Universal Robots PolyScope program: socketbuffer.urp

Program socketbuffer (installation=botross directory=/programs/APS2OsUltimosRomanticos createdIn=3.15.3.106223 lastSavedIn=3.15.3.106223 robotSerialNumber=2017357017)
Calibrated DH parameters: a=[0.0001, -0.032836, -0.39033, 0.000086, 0.000053, 0]; d=[0.089393, 264.548863, -261.578988, -2.85966, 0.094927, 0.082356]; alpha=[1.569373, -0.001603, 0.013671, 1.570599, -1.570158, 0]; deltaTheta=[0.000031, -1.49356, 1.597104, -0.103695, -0.000023, -0.000043]
Robot Program (runOnlyOnce=false)
  com_open := False
  Loop Forever
    com_open := socket_open("10.103.16.140",30000)
  Call Rotina_Contornos
SubProgram -> Rotina_Contornos
SubProgram Rotina_Pick_Caneta (keepSynchronizedWithDisk=false)
  Wait Sleep waitTime=0.01
  'a linha a seguir causa um movimento brusco e intenso'
  Script: speedl([0.5,0.5,0.5,0,0,0],0.5,5)
SubProgram Rotina_Contornos (keepSynchronizedWithDisk=false)
  'Numero de pontos em determinado segmento de contorno'
  N_pontos := socket_read_ascii_float(1)
  N := N_pontos[1]
  X := socket_read_ascii_float(N)
  Y := socket_read_ascii_float(N)
  Z := socket_read_ascii_float(N)
  Script: socket_close()
  If X[0]≠0
    pose_desejada := p[X[1]/1000,X[2]/1000,read_ascii[3]/1000,0,0,0]
    pose_atual := get_actual_tcp_pose()
    current_pose := pose_trans(Plano_BotRoss,pose_desejada)
    MoveL speed 250 mm/s, acceleration 1200 mm/s^2 (useActiveTCP=true) feature=Base
      Waypoint Waypoint (Variable): variable=current_pose
      Wait NoWait
